FUNCTION_BLOCK FB_ShortTEST2
VAR_INPUT
	execute: BOOL;
	pos2: LREAL := 2400;
END_VAR
VAR
	TIMERDONE: BOOL;
END_VAR

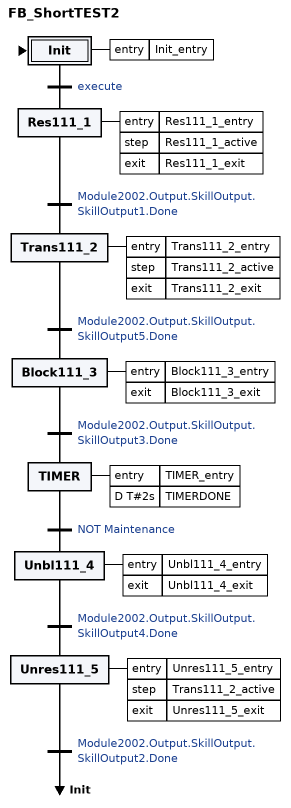
INITIAL_STEP Init:
    Init_entry(P1);  // entry action
END_STEP
TRANSITION FROM Init TO Res111_1
    := execute;
END_TRANSITION
STEP Res111_1:
    Res111_1_entry(P1);  // entry action
    Res111_1_active(N);  // step action
    Res111_1_exit(P0);  // exit action
END_STEP
TRANSITION FROM Res111_1 TO Trans111_2
    := Module2002.Output.SkillOutput.SkillOutput1.Done;
END_TRANSITION
STEP Trans111_2:
    Trans111_2_entry(P1);  // entry action
    Trans111_2_active(N);  // step action
    Trans111_2_exit(P0);  // exit action
END_STEP
TRANSITION FROM Trans111_2 TO Block111_3
    := Module2002.Output.SkillOutput.SkillOutput5.Done;
END_TRANSITION
STEP Block111_3:
    Block111_3_entry(P1);  // entry action
    Block111_3_exit(P0);  // exit action
END_STEP
TRANSITION FROM Block111_3 TO TIMER
    := Module2002.Output.SkillOutput.SkillOutput3.Done;
END_TRANSITION
STEP TIMER:
    TIMER_entry(P1);  // entry action
    TIMERDONE(D, T#2s);
END_STEP
TRANSITION FROM TIMER TO Unbl111_4
    := NOT Maintenance;
END_TRANSITION
STEP Unbl111_4:
    Unbl111_4_entry(P1);  // entry action
    Unbl111_4_exit(P0);  // exit action
END_STEP
TRANSITION FROM Unbl111_4 TO Unres111_5
    := Module2002.Output.SkillOutput.SkillOutput4.Done;
END_TRANSITION
STEP Unres111_5:
    Unres111_5_entry(P1);  // entry action
    Trans111_2_active(N);  // step action
    Unres111_5_exit(P0);  // exit action
END_STEP
TRANSITION FROM Unres111_5 TO Init
    := Module2002.Output.SkillOutput.SkillOutput2.Done;
END_TRANSITION

ACTION Res111_1_exit:
// Reservieren entry
Module2002.Input.SkillInput.SkillInput1.Execute := FALSE;
Module2002.Input.SkillInput.SkillInput1.ParameterInput.Parameterinput1.Value := 0; //TASKID
END_ACTION

ACTION Trans111_6_exit:
//TRANSPORTIEREN

Module2002.Input.SkillInput.SkillInput5.Execute := FALSE;
Module2002.Input.SkillInput.SkillInput5.ParameterInput.Parameterinput1.Value := 0; //X-Position
Module2002.Input.SkillInput.SkillInput5.ParameterInput.Parameterinput2.Value := 0; //Z-Position
Module2002.Input.SkillInput.SkillInput5.ParameterInput.Parameterinput3.Value := 0; //Velocity
Module2002.Input.SkillInput.SkillInput5.ParameterInput.Parameterinput4.Value := 0; //Acceleration
END_ACTION

ACTION Trans111_6_entry:
//TRANSPORTIEREN

Module2002.Input.SkillInput.SkillInput5.Execute := TRUE;
Module2002.Input.SkillInput.SkillInput5.ParameterInput.Parameterinput1.Value := pos2; //X-Position
Module2002.Input.SkillInput.SkillInput5.ParameterInput.Parameterinput2.Value := 80; //Z-Position
Module2002.Input.SkillInput.SkillInput5.ParameterInput.Parameterinput3.Value := 0; //Velocity
Module2002.Input.SkillInput.SkillInput5.ParameterInput.Parameterinput4.Value := 0; //Acceleration
END_ACTION

ACTION Trans111_2_entry:
//TRANSPORTIEREN

Module2002.Input.SkillInput.SkillInput5.Execute := TRUE;
Module2002.Input.SkillInput.SkillInput5.ParameterInput.Parameterinput1.Value := 1348.4; //X-Position
Module2002.Input.SkillInput.SkillInput5.ParameterInput.Parameterinput2.Value := 80; //Z-Position
Module2002.Input.SkillInput.SkillInput5.ParameterInput.Parameterinput3.Value := 0; //Velocity
Module2002.Input.SkillInput.SkillInput5.ParameterInput.Parameterinput4.Value := 0; //Acceleration
END_ACTION

ACTION Trans111_2_active:

END_ACTION

ACTION TIMER_entry:
TIMERDONE := FALSE;
END_ACTION

ACTION Unbl111_4_exit:
//unBLOCKIEREN

Module2002.Input.SkillInput.SkillInput4.Execute := FALSE; 
Module2002.Input.SkillInput.SkillInput4.ParameterInput.Parameterinput1.Value := 000; //TaskID
END_ACTION

ACTION Res111_1_active:

END_ACTION

ACTION Block111_3_exit:
//BLOCKIEREN

Module2002.Input.SkillInput.SkillInput3.Execute := FALSE;
Module2002.Input.SkillInput.SkillInput3.ParameterInput.Parameterinput1.Value := 0; //TaskID
END_ACTION

ACTION Unres111_5_entry:
//unreserve
Module2002.Input.SkillInput.SkillInput2.Execute := TRUE;
Module2002.Input.SkillInput.SkillInput2.ParameterInput.Parameterinput1.Value := 112; //TaskID
END_ACTION

ACTION Trans111_2_exit:
//TRANSPORTIEREN

Module2002.Input.SkillInput.SkillInput5.Execute := FALSE;
Module2002.Input.SkillInput.SkillInput5.ParameterInput.Parameterinput1.Value := 0; //X-Position
Module2002.Input.SkillInput.SkillInput5.ParameterInput.Parameterinput2.Value := 0; //Z-Position
Module2002.Input.SkillInput.SkillInput5.ParameterInput.Parameterinput3.Value := 0; //Velocity
Module2002.Input.SkillInput.SkillInput5.ParameterInput.Parameterinput4.Value := 0; //Acceleration
END_ACTION

ACTION Res111_1_entry:
// Reservieren entry
Module2002.Input.SkillInput.SkillInput1.Execute := TRUE;
Module2002.Input.SkillInput.SkillInput1.ParameterInput.Parameterinput1.Value := 112; //TASKID
END_ACTION

ACTION Unbl111_4_entry:
//unBLOCKIEREN

Module2002.Input.SkillInput.SkillInput4.Execute := TRUE; //FALSE weil timer
Module2002.Input.SkillInput.SkillInput4.ParameterInput.Parameterinput1.Value := 112; //TaskID
END_ACTION

ACTION Init_entry:
execute := FALSE;
END_ACTION

ACTION Block111_3_entry:
//BLOCKIEREN

Module2002.Input.SkillInput.SkillInput3.Execute := TRUE;
Module2002.Input.SkillInput.SkillInput3.ParameterInput.Parameterinput1.Value := 112; //TaskID
END_ACTION

ACTION Unres111_5_exit:
//unreserve
Module2002.Input.SkillInput.SkillInput2.Execute := FALSE;
Module2002.Input.SkillInput.SkillInput2.ParameterInput.Parameterinput1.Value := 0; //TaskID
END_ACTION

END_FUNCTION_BLOCK

(* stored: Version 1.1.0.1, ProductVersion 3.1.0.25
   POU FB_ShortTEST2: Id {e83a047a-a151-4ca8-975b-60ed0faaa80d}
   Action Res111_1_exit: Id {0448e8e5-be13-4ceb-af36-fe10a302d09e}
   Action Trans111_6_exit: Id {1634a605-8285-4caf-8480-5786436e576e}
   Action Trans111_6_entry: Id {16414cfb-ddda-4e0c-bd17-ffef1e779a23}
   Action Trans111_2_entry: Id {1b370673-6fa9-425b-a5da-b0cc70b53293}
   Action Trans111_2_active: Id {447d7ea4-5abc-4cbb-9736-5287d125a7ac}
   Action TIMER_entry: Id {497b2487-08d6-4f40-9e17-6a71558ad115}
   Action Unbl111_4_exit: Id {4cab67aa-fe03-4131-bbc0-c4ed601b9071}
   Action Res111_1_active: Id {5498b574-1c3c-4e0b-9a65-e020a83dc714}
   Action Block111_3_exit: Id {5ffca86f-f2d0-487a-a72b-bf185ceaa8a7}
   Action Unres111_5_entry: Id {6c7db6d5-6358-4e07-a2f5-6608cee285ea}
   Action Trans111_2_exit: Id {750ed05d-4ace-4f20-b558-49ef783e5504}
   Action Res111_1_entry: Id {9f4902b6-aa97-4011-a10c-ffa7624e6cd3}
   Action Unbl111_4_entry: Id {c190f06f-3fb2-4e83-9b71-fead6b2dce81}
   Action Init_entry: Id {c59b94af-47ae-4bf7-94c9-b464ae175bbf}
   Action Block111_3_entry: Id {d67e568c-47bc-4ada-9d9c-0909b77cd4bb}
   Action Unres111_5_exit: Id {dde13e88-9aad-4640-9937-6f3e9069b0a4} *)
